// TIA Portal V20 export
DATA_BLOCK "BK09"   // DB204
// stored: MemoryReserve 100
   VAR
      "X10-1 NG & MANUAL INPUT VIBRATOR-1 ON" : Bool;
      "X10-2 NG & MANUAL INPUT VIBRATOR-1 OFF" : Bool;
      "X12-1 NG & MANUAL INPUT PAD VACUUM ON" : Bool;
      "X12-2 NG & MANUAL INPUT PAD VACUUM OFF" : Bool;
      "X14-1 NG & MANUAL INPUT VIBRATOR VACUUM ON" : Bool;
      "X14-2 NG & MANUAL INPUT VIBRATOR VACUUM OFF" : Bool;
      "X16-1 NG & MANUAL INPUT VIBRATOR-2 ON" : Bool;
      "X16-2 NG & MANUAL INPUT VIBRATOR-2 OFF" : Bool;
   END_VAR
BEGIN
END_DATA_BLOCK
